{attribute addProperty BoxType "EPP2318-0001-0016"}
{attribute addProperty Id "ChannelAT %I*ARRAY[0..3] OF Channel_E4AEF59E3240Channel_1AT %Q*ARRAY[0..3] OF Channel_7F374EB03240WcStateAT %I*WcState_98A4DF7520.250InfoDataAT %I*InfoData_192954DE1620"}
{attribute addProperty CRC "4250879022"}
{attribute addProperty SizeInBites "82"}
{attribute addProperty SizeInBytes "10.25"}
TYPE EPP2318_97B4DD11 :
STRUCT
	{attribute addProperty Name "Channel"}
	Channel : ARRAY[0..3] OF Channel_E4AEF59E;
	{attribute addProperty Name "Channel_1"}
	Channel_1 : ARRAY[0..3] OF Channel_7F374EB0;
	{attribute addProperty Name "WcState"}
	WcState : WcState_98A4DF75;
	{attribute addProperty Name "InfoData"}
	InfoData : InfoData_192954DE;
END_STRUCT
END_TYPE

(* stored: Version 1.2.0.0, ProductVersion 3.1.4024.9
   DUT EPP2318_97B4DD11: Id {8df83b2c-9161-4338-bde8-addc68450122} *)
